// TIA Portal V19 export
TYPE "LEXCHANGETRAY_typeConstraintRollerEm_toHandlingXyzReq"
// stored: Access Published
   STRUCT
      transferEnable : Bool;
   END_STRUCT;
END_TYPE
